(* CODESYS project TestKlick.project

Project tree, tasks and I/O mapping:
  XV100 : XV100, Eaton Automation, version 3.5.3.0
    application Application
      libraries: Standard, 3.5.2.0 (System); TSR Libary, 1.15 (Eaton Automation)
      task Task (cyclic, interval t#10ms, priority 1) calls MAIN
      program MAIN [ST]
*)

// XV100/Application/MAIN
PROGRAM MAIN
VAR
	Execute					:BOOL;				//Startbedingung für den FB.
	x						:INT;				//Die Nummer des Com Ports.
	y						:INT;				//Wenn = 0 Wird der Port geschlossen, Wenn = 1 Wird der Port geöffnet.
												//FB Ausgänge
	Busy					:BOOL;				//Das Busy bit.
	Done					:BOOL;				//Ist 1 wenn FB fertig ist.
	State					:WORD;				//Der ENUM Wert für die ENUM Tabelle.
	Error					:BOOL;				//Ist 1 wenn es einen Error gab.	
	Klick					:FB_Click;			//Klick FB
	
//CONNECT
	Execute1				:BOOL;				//Startbedingung für den FB.
	Com1					:INT;				//Die Nummer des Com Ports.
	Port1					:BOOL;				//Wenn = 0 Wird der Port geschlossen, Wenn = 1 Wird der Port geöffnet.
												//FB Ausgänge
	Busy1					:BOOL;				//Das Busy bit.
	Done1					:BOOL;				//Ist 1 wenn FB fertig ist.
	State1					:WORD;				//Der ENUM Wert für die ENUM Tabelle.
	Error1					:BOOL;				//Ist 1 wenn es einen Error gab.	

con: Connect_with_TSR;
END_VAR

con(
	xExecute:=Execute1 , 
	iCom:=Com1 , 
	xPort:=Port1 , 
	xBusy=>Busy1 , 
	xDone=>Done1 , 
	wState=>State1 , 
	xError=>Error1 );


Klick(
	xExecute:=Execute , 
	iKlicktox:=x , 
	iKlicktoy:=y , 
	xBusy=>Busy , 
	xDone=>Done , 
	wState=>State , 
	xError=>Error );

END_PROGRAM
